PROGRAM MAIN
VAR
END_VAR

END_PROGRAM

(* stored: Version 1.1.0.1
   POU MAIN: Id {22d91436-0db9-4187-bda5-22d7266d65fa} *)
